{attribute 'qualified_only'}
{attribute 'strict'}
TYPE E_SA_CMD_TYPE :
(
	INIT := 0,	// Commands for system initialisation
	READ,		// Commands for Reading status
	CFG,		// Commands for Configuring channels
	CTRL		// Commands for Controlling positioners, e.g. CAL, REF, MOVE, STOP
);
END_TYPE

(* stored: Version 1.1.0.1, ProductVersion 3.1.4024.10
   DUT E_SA_CMD_TYPE: Id {b71ba0d7-20f0-4ea3-932a-296a0c8ec369} *)
